PROGRAM PRG_ExtractAnyStringManual
VAR
	fbExtractAnyString		: FB_ExtractAnyString;
	
	bExtractData		: BOOL;			(* set TRUE to remove prefix and suffix from strData *)
	nExtractChars		: UINT;			(* if suffix is blank, number of data chars to extract *)
	sPrefix				: T_MaxString;	(* prefix string *)
	sSuffix				: T_MaxString;	(* suffix string *)
	bIgnoreCase			: BOOL;
	eExtractMode		: E_STRING_ExtrMode	:= E_STRING_ExtrMode.WITHOUTIDENT_PURGE;

	sDataString			: T_LongSTRING;	(* string to be searched *)

	bStringFound				: BOOL;			(* TRUE = sub-string with matching prefix/suffix found *)
	sExtractedString			: T_LongSTRING;	(* extracted data *)
	nExtractedStringPos			: UDINT;			(* start pos of extracted string in strString *)
	nExtractedStringLen			: UDINT;
	nDataStringLen				: UDINT;
END_VAR

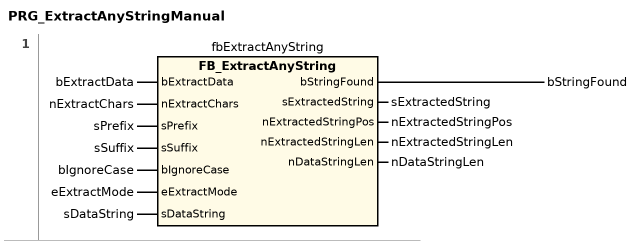
// NETWORK 1
fbExtractAnyString(
    bExtractData := bExtractData,
    nExtractChars := nExtractChars,
    sPrefix := sPrefix,
    sSuffix := sSuffix,
    bIgnoreCase := bIgnoreCase,
    eExtractMode := eExtractMode,
    sDataString := sDataString,
    sExtractedString => sExtractedString,
    nExtractedStringPos => nExtractedStringPos,
    nExtractedStringLen => nExtractedStringLen,
    nDataStringLen => nDataStringLen); // FB_ExtractAnyString
bStringFound := fbExtractAnyString.bStringFound;

END_PROGRAM

(* stored: Version 1.1.0.1
   POU PRG_ExtractAnyStringManual: Id {ee99ba5e-5d27-4821-9566-353eac5920ce}, SpecialFunc None *)
